FUNCTION fc_Hour_To_Time : Time
VAR_INPUT
		IN : REAL;
END_VAR
VAR
END_VAR

fc_Hour_To_Time := DWORD_TO_TIME(REAL_TO_DWORD(IN * 3600000));

END_FUNCTION

(* stored: Version 1.1.0.1, ProductVersion 3.1.4024.11
   POU fc_Hour_To_Time: Id {edf313fe-cd28-404e-a055-5bb8b3aa1db0}, SpecialFunc None *)
